Staubli VAL3: deutsch.dtx

public string No = "Nein"
public string Yes = "Ja "
